// TIA Portal V20 export
TYPE "type_emRelations_em6"
// stored: Access Published, Namespace Unit1
   STRUCT
      "Bool" { ExternalWritable := 'False'} : Struct
         "00" : Bool;
         "01" : Bool;
         "02" : Bool;
         "03" : Bool;
         "04" : Bool;
         "05" : Bool;
         "06" : Bool;
         "07" : Bool;
         "08" : Bool;
         "09" : Bool;
         "10" : Bool;
         "11" : Bool;
         "12" : Bool;
         "13" : Bool;
         "14" : Bool;
         "15" : Bool;
         "16" : Bool;
         "17" : Bool;
         "18" : Bool;
         "19" : Bool;
      END_STRUCT;
      LReal { ExternalWritable := 'False'} : Struct
         "00" : LReal;
         "01" : LReal;
         "02" : LReal;
         "03" : LReal;
         "04" : LReal;
         "05" : LReal;
         "06" : LReal;
         "07" : LReal;
         "08" : LReal;
         "09" : LReal;
         "10" : LReal;
         "11" : LReal;
         "12" : LReal;
         "13" : LReal;
         "14" : LReal;
         "15" : LReal;
         "16" : LReal;
         "17" : LReal;
         "18" : LReal;
         "19" : LReal;
      END_STRUCT;
      isLinked : Bool;
      state : "LUC_typeStates";
      softCam : "Unit1.type_emRelations_em6_SoftCam";
      cmStatus { S7_SetPoint := 'True'} : "Unit1.type_emRelations_em6_cmStatus";
      sequence { S7_SetPoint := 'True'} : "Unit1.type_emRelations_em6_sequence";
   END_STRUCT;
END_TYPE
